{attribute 'GeneratedUsingTerminal: EL9222-4433-0018'}
{attribute addProperty BoxType "EL9222-4433-0018"}
{attribute addProperty Id "ControlAT %Q*Control_534FEB192"}
{attribute addProperty CRC "16861492"}
{attribute addProperty Size "2"}
TYPE OCP_Outputs_Channel_01014934 EXTENDS OutputBase_10CEE7DE :
STRUCT
	{attribute addProperty Name "Control"}
	Control AT %Q* : Control_534FEB19;
END_STRUCT
END_TYPE

(* stored: Version 1.2.0.0, ProductVersion 3.1.4024.11
   DUT OCP_Outputs_Channel_01014934: Id {0a513ad5-bcad-400c-b8d3-e89c52c60852} *)
